{attribute 'qualified_only'}
VAR_GLOBAL
	//DataSources
	//Live:
	fbT1_InputSource: FB_T1_InputSource;
	//Historical:
	//Empty:
	
	fbT1_IecCriticalSection: FB_IecCriticalSection;
	
	//Historical DataSource parameter
	nHistMaxInputBuffer: UDINT := 100;
	nHistMaxSampleCount: UDINT := 100;
	
	stReset: ST_AnalysisReset;
	
	//Scope ADS Push Target NetID
	sScopeServerNetID: T_AmsNetID := '10.123.65.55.1.1';
END_VAR

(* stored: GVL Analytics: Id 19d082b0-3e05-4c8e-be7e-bd53966b1692 *)
